# EPICS substitutions: iocBoot/ioc14lab/iocEnvVar.substitutions
#==============================================================================
#
# Abs:  IOC Administration Records
#
# Name: iocAdmin.substitutions
#
#==============================================================================
# Edited to work at BioCARS.

file "$(DEVIOCSTATS)/iocAdminLib/Db/iocEnvVar.db"
{
pattern { IOCNAME, ENVNAME      , ENVVAR                          , ENVTYPE}
	{ 14IDB , LOCATION     , LOCATION                        , env    }
	{ 14IDB , ENGINEER     , ENGINEER                        , env    }
	{ 14IDB , CA_ADDR_LIST , EPICS_CA_ADDR_LIST              , epics  }
	{ 14IDB , CA_CONN_TIME , EPICS_CA_CONN_TMO               , epics  }
	{ 14IDB , CA_AUTO_ADDR , EPICS_CA_AUTO_ADDR_LIST         , epics  }
	{ 14IDB , CA_RPTR_PORT , EPICS_CA_REPEATER_PORT          , epics  }
	{ 14IDB , CA_SRVR_PORT , EPICS_CA_SERVER_PORT            , epics  }
	{ 14IDB , CA_MAX_ARRAY , EPICS_CA_MAX_ARRAY_BYTES        , epics  }
	{ 14IDB , CA_SRCH_TIME , EPICS_CA_MAX_SEARCH_PERIOD      , epics  }
	{ 14IDB , CA_BEAC_TIME , EPICS_CA_BEACON_PERIOD          , epics  }
	{ 14IDB , TIMEZONE     , EPICS_TIMEZONE                  , epics  }
	{ 14IDB , TS_NTP_INET  , EPICS_TS_NTP_INET               , epics  }
	{ 14IDB , IOC_LOG_PORT , EPICS_IOC_LOG_PORT              , epics  }
	{ 14IDB , IOC_LOG_INET , EPICS_IOC_LOG_INET              , epics  }
}
